# EPICS substitutions: asubtest-mk-IOCApp/Db/userHostlinux.substitutions
# Example substitutions file

#file "db/asub.db" {
#    { user = "mrippaHost" }
#
#}

file db/asub4.db {
    pattern { user, no, scan }
        { "lnx", 2, "Passive" }
}
